// Mitsubishi GX Works2 project: e03   PLC: Q02/Q02H

PROGRAM MAIN
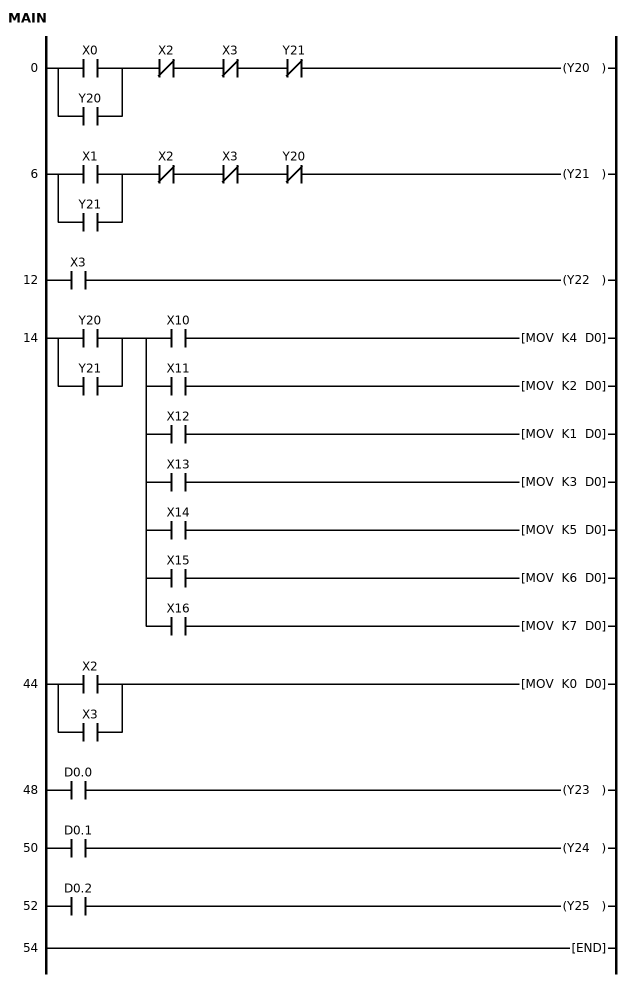
0     LD      X0
      OR      Y20
      ANI     X2
      ANI     X3
      ANI     Y21
      OUT     Y20
6     LD      X1
      OR      Y21
      ANI     X2
      ANI     X3
      ANI     Y20
      OUT     Y21
12    LD      X3
      OUT     Y22
14    LD      Y20
      OR      Y21
      MPS
      AND     X10
      MOV     K4 D0
      MRD
      AND     X11
      MOV     K2 D0
      MRD
      AND     X12
      MOV     K1 D0
      MRD
      AND     X13
      MOV     K3 D0
      MRD
      AND     X14
      MOV     K5 D0
      MRD
      AND     X15
      MOV     K6 D0
      MPP
      AND     X16
      MOV     K7 D0
44    LD      X2
      OR      X3
      MOV     K0 D0
48    LD      D0.0
      OUT     Y23
50    LD      D0.1
      OUT     Y24
52    LD      D0.2
      OUT     Y25
54    END
END_PROGRAM
